{attribute addProperty BoxType "EL3773-0000-0018"}
{attribute addProperty Id "U3_StatusAT %I*U3_Status_E2EFACF1162"}
{attribute addProperty CRC "493146806"}
{attribute addProperty SizeInBites "16"}
{attribute addProperty SizeInBytes "2"}
TYPE L3_Voltage_Status_1D64D2B6 :
STRUCT
	{attribute addProperty Name "U3_Status"}
	U3_Status AT %I* : U3_Status_E2EFACF1;
END_STRUCT
END_TYPE

(* stored: Version 1.2.0.0, ProductVersion 3.1.4024.9
   DUT L3_Voltage_Status_1D64D2B6: Id {179dbfc8-4e20-414b-85e0-871fb22c670a} *)
